{attribute 'pack_mode' := '1'} 
// ------------------------------------------------------------------------- 
//  SRCI Robot Library                                                
// ------------------------------------------------------------------------- 
//                                                                           
//  Object:      TelegramRobToPlcCyclicOptionalCartesianPosExt                                       
//  Author:      Thorsten Brach                                                
//  Date:        2024-06-01
//
//  Description:                                              
//   
//                                                                           
//  Copyright: 
//    (C) 2024 Thorsten Brach. All rights reserved                                                                         
//                                                                           
//  Disclaimer:                                                                           
//    This project is provided without any guarantee and can be used for   
//    private and commercial purposes. Any commercial use is at the user’s 
//    own risk and responsibility.
//
// -------------------------------------------------------------------------
TYPE TelegramRobToPlcCyclicOptionalCartesianPositionExt :
STRUCT
  /// Position of second external axis
  E2 : REAL;
  /// Position of third external axis
  E3 : REAL;
  /// Position of fourth external axis
  E4 : REAL;
  /// Position of fifth external axis
  E5 : REAL;
  /// Position of sixth external axis
  E6 : REAL;    
END_STRUCT
END_TYPE

{attribute 'pack_mode' := '1'} 
// ------------------------------------------------------------------------- 
//  SRCI Robot Library                                                
// ------------------------------------------------------------------------- 
//                                                                           
//  Object:      TelegramRobToPlcCyclicOptionalCurrent                                       
//  Author:      Thorsten Brach                                                
//  Date:        2024-06-01
//
//  Description:                                              
//   
//                                                                           
//  Copyright: 
//    (C) 2024 Thorsten Brach. All rights reserved                                                                         
//                                                                           
//  Disclaimer:                                                                           
//    This project is provided without any guarantee and can be used for   
//    private and commercial purposes. Any commercial use is at the user’s 
//    own risk and responsibility.
//
// -------------------------------------------------------------------------
TYPE TelegramRobToPlcCyclicOptionalCurrent :
STRUCT
  /// Current of first joint of the robot
  J1 : REAL;
  /// Current of second joint of the robot
  J2 : REAL;
  /// Current of third joint of the robot
  J3 : REAL;
  /// Current of fourth joint of the robot
  J4 : REAL;
  /// Current of fifth joint of the robot
  J5 : REAL;
  /// Current of sixth joint of the robot
  J6 : REAL;  
END_STRUCT
END_TYPE

{attribute 'pack_mode' := '1'} 
// ------------------------------------------------------------------------- 
//  SRCI Robot Library                                                
// ------------------------------------------------------------------------- 
//                                                                           
//  Object:      TelegramRobToPlcCyclicOptionalCurrentExt                                       
//  Author:      Thorsten Brach                                                
//  Date:        2024-06-01
//
//  Description:                                              
//   
//                                                                           
//  Copyright: 
//    (C) 2024 Thorsten Brach. All rights reserved                                                                         
//                                                                           
//  Disclaimer:                                                                           
//    This project is provided without any guarantee and can be used for   
//    private and commercial purposes. Any commercial use is at the user’s 
//    own risk and responsibility.
//
// -------------------------------------------------------------------------
TYPE TelegramRobToPlcCyclicOptionalCurrentExt :
STRUCT
  /// Current of first external joint of the robot
  E1 : REAL;
  /// Current of second external axis
  E2: REAL;
  /// Current of third external axis
  E3: REAL;
  /// Current of fourth external axis
  E4: REAL;
  /// Current of fifth external axis
  E5: REAL;
  /// Current of sixth external axis
  E6: REAL;  
END_STRUCT
END_TYPE

{attribute 'pack_mode' := '1'} 
// ------------------------------------------------------------------------- 
//  SRCI Robot Library                                                
// ------------------------------------------------------------------------- 
//                                                                           
//  Object:      TelegramRobToPlcCyclicOptionalForce                                       
//  Author:      Thorsten Brach                                                
//  Date:        2024-06-01
//
//  Description:                                              
//   
//                                                                           
//  Copyright: 
//    (C) 2024 Thorsten Brach. All rights reserved                                                                         
//                                                                           
//  Disclaimer:                                                                           
//    This project is provided without any guarantee and can be used for   
//    private and commercial purposes. Any commercial use is at the user’s 
//    own risk and responsibility.
//
// -------------------------------------------------------------------------
TYPE TelegramRobToPlcCyclicOptionalForce :
STRUCT
  /// Force on the X-Axis
  X : REAL;
  /// Force on the Y-Axis
  Y : REAL;
  /// Force on the Z-Axis
  Z : REAL;
  /// Force around the X-Axis (RX)
  Rx : REAL;
  /// Force around the Y-Axis (RY)
  Ry : REAL;
  /// Force around the Z-Axis (RZ)
  Rz : REAL;
END_STRUCT
END_TYPE

{attribute 'pack_mode' := '1'} 
// ------------------------------------------------------------------------- 
//  SRCI Robot Library                                                
// ------------------------------------------------------------------------- 
//                                                                           
//  Object:      TelegramRobToPlcCyclicOptionalForceExt                                       
//  Author:      Thorsten Brach                                                
//  Date:        2024-06-01
//
//  Description:                                              
//   
//                                                                           
//  Copyright: 
//    (C) 2024 Thorsten Brach. All rights reserved                                                                         
//                                                                           
//  Disclaimer:                                                                           
//    This project is provided without any guarantee and can be used for   
//    private and commercial purposes. Any commercial use is at the user’s 
//    own risk and responsibility.
//
// -------------------------------------------------------------------------
TYPE TelegramRobToPlcCyclicOptionalForceExt :
STRUCT
  /// Force on the external axis 1
  E1 : REAL;
  /// Force on the external axis 2
  E2 : REAL;
  /// Force on the external axis 3
  E3 : REAL;
  /// Force om the external axis 4
  E4 : REAL;
  /// Force on the external axis 5
  E5 : REAL;
  /// Force on the external axis 6
  E6 : REAL;
END_STRUCT
END_TYPE

{attribute 'pack_mode' := '1'} 
// ------------------------------------------------------------------------- 
//  SRCI Robot Library                                                
// ------------------------------------------------------------------------- 
//                                                                           
//  Object:      TelegramRobToPlcCyclicOptionalJointPosition                                       
//  Author:      Thorsten Brach                                                
//  Date:        2024-06-01
//
//  Description:                                              
//   
//                                                                           
//  Copyright: 
//    (C) 2024 Thorsten Brach. All rights reserved                                                                         
//                                                                           
//  Disclaimer:                                                                           
//    This project is provided without any guarantee and can be used for   
//    private and commercial purposes. Any commercial use is at the user’s 
//    own risk and responsibility.
//
// -------------------------------------------------------------------------
TYPE TelegramRobToPlcCyclicOptionalJointPosition :
STRUCT
  /// Position of first joint of the robot
  J1 : REAL;
  /// Position of second joint of the robot
  J2 : REAL;
  /// Position of third joint of the robot
  J3 : REAL;
  /// Position of fourth joint of the robot
  J4 : REAL;
  /// Position of fifth joint of the robot
  J5 : REAL;
  /// Position of sixth joint of the robot
  J6 : REAL;
  /// Position of first external axis 
  E1 : REAL;  
  /// Reserve
  E1_Reserve : WORD;
END_STRUCT
END_TYPE

{attribute 'pack_mode' := '1'} 
// ------------------------------------------------------------------------- 
//  SRCI Robot Library                                                
// ------------------------------------------------------------------------- 
//                                                                           
//  Object:      TelegramRobToPlcCyclicOptionalJointPositionExt                                       
//  Author:      Thorsten Brach                                                
//  Date:        2024-06-01
//
//  Description:                                              
//   
//                                                                           
//  Copyright: 
//    (C) 2024 Thorsten Brach. All rights reserved                                                                         
//                                                                           
//  Disclaimer:                                                                           
//    This project is provided without any guarantee and can be used for   
//    private and commercial purposes. Any commercial use is at the user’s 
//    own risk and responsibility.
//
// -------------------------------------------------------------------------
TYPE TelegramRobToPlcCyclicOptionalJointPositionExt :
STRUCT
  /// Position of second external axis
  E2: REAL;
  /// Position of third external axis
  E3: REAL;
  /// Position of fourth external axis
  E4: REAL;
  /// Position of fifth external axis
  E5: REAL;
  /// Position of sixth external axis
  E6: REAL;    
END_STRUCT
END_TYPE

{attribute 'pack_mode' := '1'} 
// ------------------------------------------------------------------------- 
//  SRCI Robot Library                                                
// ------------------------------------------------------------------------- 
//                                                                           
//  Object:      TelegramRobToPlcCyclicOptionalSubProgramData                                       
//  Author:      Thorsten Brach                                                
//  Date:        2024-06-01
//
//  Description:                                              
//   
//                                                                           
//  Copyright: 
//    (C) 2024 Thorsten Brach. All rights reserved                                                                         
//                                                                           
//  Disclaimer:                                                                           
//    This project is provided without any guarantee and can be used for   
//    private and commercial purposes. Any commercial use is at the user’s 
//    own risk and responsibility.
//
// -------------------------------------------------------------------------
TYPE TelegramRobToPlcCyclicOptionalSubProgramData :
STRUCT
  /// Sub program data
  Data : ARRAY [0..25] OF BYTE;
END_STRUCT
END_TYPE

{attribute 'pack_mode' := '1'} 
// ------------------------------------------------------------------------- 
//  SRCI Robot Library                                                
// ------------------------------------------------------------------------- 
//                                                                           
//  Object:      ActivateNextCommandOutCmd                                       
//  Author:      Thorsten Brach                                                
//  Date:        2024-06-01
//
//  Description:                                              
//   
//                                                                           
//  Copyright: 
//    (C) 2024 Thorsten Brach. All rights reserved                                                                         
//                                                                           
//  Disclaimer:                                                                           
//    This project is provided without any guarantee and can be used for   
//    private and commercial purposes. Any commercial use is at the user’s 
//    own risk and responsibility.
//
// -------------------------------------------------------------------------
TYPE ActivateNextCommandOutCmd :
STRUCT
  /// Unique system-generated ID of the "Action" when the function is triggered.
  /// • >0: The "Action" is started by the trigger function with identical FollowID.
  /// • <0: The "Action" is stopped by the trigger function with identical FollowID.
  /// For more information see chapter 5.5.12.4 EmitterID, ListenerID, FollowID and OriginID
  OriginID           : INT;
  /// Relates to ListenerID >0
  /// Number of successful trigger -based command invocations
  /// For more information refer to chapter 5.5.12.4.
  InvocationCounter  : USINT;
END_STRUCT
END_TYPE

{attribute 'pack_mode' := '1'} 
// ------------------------------------------------------------------------- 
//  SRCI Robot Library                                                
// ------------------------------------------------------------------------- 
//                                                                           
//  Object:      ActivateNextCommandParCmd                                       
//  Author:      Thorsten Brach                                                
//  Date:        2024-06-01
//
//  Description:                                              
//   
//                                                                           
//  Copyright: 
//    (C) 2024 Thorsten Brach. All rights reserved                                                                         
//                                                                           
//  Disclaimer:                                                                           
//    This project is provided without any guarantee and can be used for   
//    private and commercial purposes. Any commercial use is at the user’s 
//    own risk and responsibility.
//
// -------------------------------------------------------------------------
TYPE ActivateNextCommandParCmd :
STRUCT
  /// Processing mode
  ProcessingMode : ProcessingMode;
  /// ID of the trigger function that may be triggered:
  /// • 0: Immediately (default). - Start executing THIS function immediately.
  /// • >0: Triggero Start executing when the trigger function with the identical EmitterID is called.
  /// For more information see chapter 5.5.12.4.
  ListenerID     : SINT;
END_STRUCT
END_TYPE

{attribute 'pack_mode' := '1'} 
// ------------------------------------------------------------------------- 
//  SRCI Robot Library                                                
// ------------------------------------------------------------------------- 
//                                                                           
//  Object:      ActivateNextCommandRecvData                                       
//  Author:      Thorsten Brach                                                
//  Date:        2024-06-01
//
//  Description:                                              
//   
//                                                                           
//  Copyright: 
//    (C) 2024 Thorsten Brach. All rights reserved                                                                         
//                                                                           
//  Disclaimer:                                                                           
//    This project is provided without any guarantee and can be used for   
//    private and commercial purposes. Any commercial use is at the user’s 
//    own risk and responsibility.
//
// -------------------------------------------------------------------------
TYPE ActivateNextCommandRecvData EXTENDS RspHeader :
STRUCT
  /// Relates to ListenerID >0
  /// Number of successful trigger -based command invocations
  /// For more information refer to chapter 5.5.12.4.
  InvocationCounter  : USINT;
  /// Reserve
  Reserve            : SINT;
  /// Unique system-generated ID of the "Action" when the function is triggered.
  /// • >0: The "Action" is started by the trigger function with identical FollowID.
  /// • <0: The "Action" is stopped by the trigger function with identical FollowID.
  /// For more information see chapter 5.5.12.4 EmitterID, ListenerID, FollowID and OriginID
  OriginID           : INT;
END_STRUCT
END_TYPE

{attribute 'pack_mode' := '1'}
// ------------------------------------------------------------------------- 
//  SRCI Robot Library                                                
// ------------------------------------------------------------------------- 
//                                                                           
//  Object:      ActivateNextCommandParCmd                                       
//  Author:      Thorsten Brach                                                
//  Date:        2024-06-01
//
//  Description:                                              
//   
//                                                                           
//  Copyright: 
//    (C) 2024 Thorsten Brach. All rights reserved                                                                         
//                                                                           
//  Disclaimer:                                                                           
//    This project is provided without any guarantee and can be used for   
//    private and commercial purposes. Any commercial use is at the user’s 
//    own risk and responsibility.
//
// -------------------------------------------------------------------------
TYPE ActivateNextCommandSendData EXTENDS CmdHeader:   
STRUCT  
  /// ID of Action that will be executed when this command is active
  /// • >0: Start Action        - Start executing the Action function with the identical ListenerID.
  /// • <0: Stop Action         - Stop executing the Action function with the identical ListenerID.
  /// •  0: Undefined (default) - If no EmitterID is defined, the function returns an error message
  /// For more information see chapter 5.5.12.4
  EmitterID  : ARRAY[0..3] OF SINT;  
  /// ID of the trigger function that may be triggered:
  /// • 0: Immediately (default). - Start executing THIS function immediately.
  /// • >0: Triggero Start executing when the trigger function with the identical EmitterID is called.
  /// For more information see chapter 5.5.12.4.
  ListenerID : SINT;
  /// Reserve
  Reserve    : BYTE;
END_STRUCT
END_TYPE

{attribute 'pack_mode' := '1'} 
// ------------------------------------------------------------------------- 
//  SRCI Robot Library                                                
// ------------------------------------------------------------------------- 
//                                                                           
//  Object:      ActivateWorkAreaOutCmd                                       
//  Author:      Thorsten Brach                                                
//  Date:        2024-06-01
//
//  Description:                                              
//   
//                                                                           
//  Copyright: 
//    (C) 2024 Thorsten Brach. All rights reserved                                                                         
//                                                                           
//  Disclaimer:                                                                           
//    This project is provided without any guarantee and can be used for   
//    private and commercial purposes. Any commercial use is at the user’s 
//    own risk and responsibility.
//
// -------------------------------------------------------------------------
TYPE ActivateWorkAreaOutCmd :
STRUCT
END_STRUCT
END_TYPE

{attribute 'pack_mode' := '1'} 
// ------------------------------------------------------------------------- 
//  SRCI Robot Library                                                
// ------------------------------------------------------------------------- 
//                                                                           
//  Object:      ActivateWorkAreaParCmd                                       
//  Author:      Thorsten Brach                                                
//  Date:        2024-06-01
//
//  Description:                                              
//   
//                                                                           
//  Copyright: 
//    (C) 2024 Thorsten Brach. All rights reserved                                                                         
//                                                                           
//  Disclaimer:                                                                           
//    This project is provided without any guarantee and can be used for   
//    private and commercial purposes. Any commercial use is at the user’s 
//    own risk and responsibility.
//
// -------------------------------------------------------------------------
TYPE ActivateWorkAreaParCmd :
STRUCT
  /// Index of the robot work area to be activated
  /// • 0 (default)..254
  WorkAreaNo         : USINT;
  /// Set to activate work area defined by Index.
  /// Reset to deactivate work area defined by Index.
  ActivateArea       : BOOL;
END_STRUCT
END_TYPE

{attribute 'pack_mode' := '1'} 
// ------------------------------------------------------------------------- 
//  SRCI Robot Library                                                
// ------------------------------------------------------------------------- 
//                                                                           
//  Object:      ActivateWorkAreaRecvData                                       
//  Author:      Thorsten Brach                                                
//  Date:        2024-06-01
//
//  Description:                                              
//   
//                                                                           
//  Copyright: 
//    (C) 2024 Thorsten Brach. All rights reserved                                                                         
//                                                                           
//  Disclaimer:                                                                           
//    This project is provided without any guarantee and can be used for   
//    private and commercial purposes. Any commercial use is at the user’s 
//    own risk and responsibility.
//
// -------------------------------------------------------------------------
TYPE ActivateWorkAreaRecvData EXTENDS RspHeader :
STRUCT
END_STRUCT
END_TYPE

{attribute 'pack_mode' := '1'}
// ------------------------------------------------------------------------- 
//  SRCI Robot Library                                                
// ------------------------------------------------------------------------- 
//                                                                           
//  Object:      ActivateWorkAreaParCmd                                       
//  Author:      Thorsten Brach                                                
//  Date:        2024-06-01
//
//  Description:                                              
//   
//                                                                           
//  Copyright: 
//    (C) 2024 Thorsten Brach. All rights reserved                                                                         
//                                                                           
//  Disclaimer:                                                                           
//    This project is provided without any guarantee and can be used for   
//    private and commercial purposes. Any commercial use is at the user’s 
//    own risk and responsibility.
//
// -------------------------------------------------------------------------
TYPE ActivateWorkAreaSendData EXTENDS CmdHeader:   
STRUCT  
  /// Index of the robot work area to be activated
  /// • 0 (default)..254
  WorkAreaNo         : USINT;
  /// Set to activate work area defined by Index.
  /// Reset to deactivate work area defined by Index.
  ActivateArea       : BOOL;
END_STRUCT
END_TYPE

{attribute 'pack_mode' := '1'} 
// ------------------------------------------------------------------------- 
//  SRCI Robot Library                                                
// ------------------------------------------------------------------------- 
//                                                                           
//  Object:      BrakeTestOutCmd                                       
//  Author:      Thorsten Brach                                                
//  Date:        2024-06-01
//
//  Description:                                              
//   
//                                                                           
//  Copyright: 
//    (C) 2024 Thorsten Brach. All rights reserved                                                                         
//                                                                           
//  Disclaimer:                                                                           
//    This project is provided without any guarantee and can be used for   
//    private and commercial purposes. Any commercial use is at the user’s 
//    own risk and responsibility.
//
// -------------------------------------------------------------------------
TYPE BrakeTestOutCmd :
STRUCT
  /// Indicates the result of the brake test of the robot axes related to the brake test.
  /// • TRUE: The brake test has been realized successfully.
  /// • FALSE: The brake test failed. 
  /// See Table 6-735 for bit assignment.
  RobotAxesStatus    : RobotAxesFlags;
  /// Indicates the result of the brake test of the external robot axes related to the brake test.
  /// • TRUE: The brake test has been realized successfully.
  /// • FALSE: The brake test failed.
  /// See Table 6-735 for bit assignment.
  ExternalAxesStatus : ExternalAxesFlags;
  /// Indicates the warning messages availability related to the brake functionality of the robot axes reported by the RC.
  /// • TRUE: One or more warning messages are available.
  /// • FALSE: No warning message is available.
  /// See Table 6-735 for bit assignment.
  RobotAxesWarning   : RobotAxesFlags;
  /// Indicates the warning messages availability related to the brake functionality of the external robot axis reported by the RC.
  /// • TRUE: One or more warning messages are available.
  /// • FALSE: No warning message is available.
  /// See Table 6-735 for bit assignment.
  ExternalAxesWarning: ExternalAxesFlags;
END_STRUCT
END_TYPE

{attribute 'pack_mode' := '1'} 
// ------------------------------------------------------------------------- 
//  SRCI Robot Library                                                
// ------------------------------------------------------------------------- 
//                                                                           
//  Object:      BrakeTestParCmd                                       
//  Author:      Thorsten Brach                                                
//  Date:        2024-06-01
//
//  Description:                                              
//   
//                                                                           
//  Copyright: 
//    (C) 2024 Thorsten Brach. All rights reserved                                                                         
//                                                                           
//  Disclaimer:                                                                           
//    This project is provided without any guarantee and can be used for   
//    private and commercial purposes. Any commercial use is at the user’s 
//    own risk and responsibility.
//
// -------------------------------------------------------------------------
TYPE BrakeTestParCmd :
STRUCT
  /// Parameter which determines the behavior towards the previously sent and still active or buffered commands.
  AbortingMode       : AbortingMode;
  /// Defines which of the robot axis should be activated for the brake test.
  /// • TRUE (default): Axis activated.
  /// • FALSE: Axis deactivated.
  /// See Table 6-735 for bit assignment.
  RobotAxesActive    : RobotAxesFlags;
  /// Defines which of the external robot axis should be activated for the brake test.
  /// • TRUE: Axis activated.
  /// • FALSE (default): Axis deactivated.
  /// See Table 6-735 for bit assignment.   
  ExternalAxesActive : ExternalAxesFlags;
  /// Defines the target sequence in which the command will be executed
  SequenceFlag       : SequenceFlag;
END_STRUCT
END_TYPE

{attribute 'pack_mode' := '1'} 
// ------------------------------------------------------------------------- 
//  SRCI Robot Library                                                
// ------------------------------------------------------------------------- 
//                                                                           
//  Object:      BrakeTestRecvData                                       
//  Author:      Thorsten Brach                                                
//  Date:        2024-06-01
//
//  Description:                                              
//   
//                                                                           
//  Copyright: 
//    (C) 2024 Thorsten Brach. All rights reserved                                                                         
//                                                                           
//  Disclaimer:                                                                           
//    This project is provided without any guarantee and can be used for   
//    private and commercial purposes. Any commercial use is at the user’s 
//    own risk and responsibility.
//
// -------------------------------------------------------------------------
TYPE BrakeTestRecvData EXTENDS RspHeader :
STRUCT
  /// Indicates the result of the brake test of the robot axes related to the brake test.
  /// • TRUE: The brake test has been realized successfully.
  /// • FALSE: The brake test failed. 
  /// See Table 6-735 for bit assignment.
  RobotAxesStatus    : BYTE;
  /// Indicates the result of the brake test of the external robot axes related to the brake test.
  /// • TRUE: The brake test has been realized successfully.
  /// • FALSE: The brake test failed.
  /// See Table 6-735 for bit assignment.
  ExternalAxesStatus : BYTE;
  /// Indicates the warning messages availability related to the brake functionality of the robot axes reported by the RC.
  /// • TRUE: One or more warning messages are available.
  /// • FALSE: No warning message is available.
  /// See Table 6-735 for bit assignment.
  RobotAxesWarning   : BYTE;
  /// Indicates the warning messages availability related to the brake functionality of the external robot axis reported by the RC.
  /// • TRUE: One or more warning messages are available.
  /// • FALSE: No warning message is available.
  /// See Table 6-735 for bit assignment.
  ExternalAxesWarning: BYTE;
END_STRUCT
END_TYPE

{attribute 'pack_mode' := '1'}
// ------------------------------------------------------------------------- 
//  SRCI Robot Library                                                
// ------------------------------------------------------------------------- 
//                                                                           
//  Object:      BrakeTestSendData                                       
//  Author:      Thorsten Brach                                                
//  Date:        2024-06-01
//
//  Description:                                              
//   
//                                                                           
//  Copyright: 
//    (C) 2024 Thorsten Brach. All rights reserved                                                                         
//                                                                           
//  Disclaimer:                                                                           
//    This project is provided without any guarantee and can be used for   
//    private and commercial purposes. Any commercial use is at the user’s 
//    own risk and responsibility.
//
// -------------------------------------------------------------------------
TYPE BrakeTestSendData EXTENDS CmdHeader:   
STRUCT
  /// Defines which of the robot axis should be activated for the brake test.
  /// • TRUE (default): Axis activated.
  /// • FALSE: Axis deactivated.
  /// See Table 6-735 for bit assignment.
  RobotAxesActive    : BYTE;
  /// Defines which of the external robot axis should be activated for the brake test.
  /// • TRUE: Axis activated.
  /// • FALSE (default): Axis deactivated.
  /// See Table 6-735 for bit assignment.   
  ExternalAxesActive : BYTE; 
END_STRUCT
END_TYPE

{attribute 'pack_mode' := '1'} 
// ------------------------------------------------------------------------- 
//  SRCI Robot Library                                                
// ------------------------------------------------------------------------- 
//                                                                           
//  Object:      BrakeTestOutCmd                                       
//  Author:      Thorsten Brach                                                
//  Date:        2024-06-01
//
//  Description:                                              
//   
//                                                                           
//  Copyright: 
//    (C) 2024 Thorsten Brach. All rights reserved                                                                         
//                                                                           
//  Disclaimer:                                                                           
//    This project is provided without any guarantee and can be used for   
//    private and commercial purposes. Any commercial use is at the user’s 
//    own risk and responsibility.
//
// -------------------------------------------------------------------------
TYPE OpenBrakeOutCmd :
STRUCT
  /// TRUE when "OpenBrake" is active.
  Enabled                   : BOOL;  
  /// Indicates the brake release status of the main robot axes.
  /// • TRUE: The brake of the axis is opened.
  /// • FALSE: The brake of the axis is closed.
  /// See Table 6-735 for bit assignment
  RobotAxesBrakeReleased    : RobotAxesFlags;
  /// Indicates the brake release status of the external robot axes.
  /// • TRUE: The brake of the axis is opened.
  /// • FALSE: The brake of the axis is closed/not supported
  /// See Table 6-735 for bit assignment
  ExternalAxesBrakeReleased : ExternalAxesFlags;
END_STRUCT
END_TYPE

{attribute 'pack_mode' := '1'} 
// ------------------------------------------------------------------------- 
//  SRCI Robot Library                                                
// ------------------------------------------------------------------------- 
//                                                                           
//  Object:      OpenBrakeParCmd                                       
//  Author:      Thorsten Brach                                                
//  Date:        2024-06-01
//
//  Description:                                              
//   
//                                                                           
//  Copyright: 
//    (C) 2024 Thorsten Brach. All rights reserved                                                                         
//                                                                           
//  Disclaimer:                                                                           
//    This project is provided without any guarantee and can be used for   
//    private and commercial purposes. Any commercial use is at the user’s 
//    own risk and responsibility.
//
// -------------------------------------------------------------------------
TYPE OpenBrakeParCmd :
STRUCT
  /// Defines which brake of the robot axes must be released.
  /// • TRUE: Open the brake of the axis.
  /// • FALSE (default): Close the brake of the axis.
  RobotAxesBrakeRelease    : RobotAxesFlags;
  /// Defines which brake of the external robot axis must be released.
  /// • TRUE: Open the brake of the axis.
  /// • FALSE (default): Close the brake of the axis.
  /// See Table 6-676 for bit assignment.
  ExternalAxesBrakeRelease : ExternalAxesFlags;
END_STRUCT
END_TYPE

{attribute 'pack_mode' := '1'} 
// ------------------------------------------------------------------------- 
//  SRCI Robot Library                                                
// ------------------------------------------------------------------------- 
//                                                                           
//  Object:      BrakeTestRecvData                                       
//  Author:      Thorsten Brach                                                
//  Date:        2024-06-01
//
//  Description:                                              
//   
//                                                                           
//  Copyright: 
//    (C) 2024 Thorsten Brach. All rights reserved                                                                         
//                                                                           
//  Disclaimer:                                                                           
//    This project is provided without any guarantee and can be used for   
//    private and commercial purposes. Any commercial use is at the user’s 
//    own risk and responsibility.
//
// -------------------------------------------------------------------------
TYPE OpenBrakeRecvData EXTENDS RspHeader :
STRUCT
  /// TRUE when "OpenBrake" is active.
  Enabled                   : BYTE;  
  /// Indicates the brake release status of the main robot axes.
  /// • TRUE: The brake of the axis is opened.
  /// • FALSE: The brake of the axis is closed.
  /// See Table 6-735 for bit assignment
  RobotAxesBrakeReleased    : BYTE;
  /// Indicates the brake release status of the external robot axes.
  /// • TRUE: The brake of the axis is opened.
  /// • FALSE: The brake of the axis is closed/not supported
  /// See Table 6-735 for bit assignment
  ExternalAxesBrakeReleased : BYTE;
END_STRUCT
END_TYPE

{attribute 'pack_mode' := '1'}
// ------------------------------------------------------------------------- 
//  SRCI Robot Library                                                
// ------------------------------------------------------------------------- 
//                                                                           
//  Object:      BrakeTestSendData                                       
//  Author:      Thorsten Brach                                                
//  Date:        2024-06-01
//
//  Description:                                              
//   
//                                                                           
//  Copyright: 
//    (C) 2024 Thorsten Brach. All rights reserved                                                                         
//                                                                           
//  Disclaimer:                                                                           
//    This project is provided without any guarantee and can be used for   
//    private and commercial purposes. Any commercial use is at the user’s 
//    own risk and responsibility.
//
// -------------------------------------------------------------------------
TYPE OpenBrakeSendData EXTENDS CmdHeader:   
STRUCT
  /// Defines which brake of the robot axes must be released.
  /// • TRUE: Open the brake of the axis.
  /// • FALSE (default): Close the brake of the axis.
  RobotAxesBrakeRelease    : BYTE;
  /// Defines which brake of the external robot axis must be released.
  /// • TRUE: Open the brake of the axis.
  /// • FALSE (default): Close the brake of the axis.
  /// See Table 6-676 for bit assignment.
  ExternalAxesBrakeRelease : BYTE;
END_STRUCT
END_TYPE

{attribute 'pack_mode' := '1'} 
// ------------------------------------------------------------------------- 
//  SRCI Robot Library                                                
// ------------------------------------------------------------------------- 
//                                                                           
//  Object:      EnableRobotOutCmd                                       
//  Author:      Thorsten Brach                                                
//  Date:        2024-06-01
//
//  Description:                                              
//   
//                                                                           
//  Copyright: 
//    (C) 2024 Thorsten Brach. All rights reserved                                                                         
//                                                                           
//  Disclaimer:                                                                           
//    This project is provided without any guarantee and can be used for   
//    private and commercial purposes. Any commercial use is at the user’s 
//    own risk and responsibility.
//
// -------------------------------------------------------------------------
TYPE EnableRobotOutCmd :
STRUCT
  /// TRUE when robot is set to RA power state "Enabled"
  Enabled           : BOOL;
END_STRUCT
END_TYPE

{attribute 'pack_mode' := '1'} 
// ------------------------------------------------------------------------- 
//  SRCI Robot Library                                                
// ------------------------------------------------------------------------- 
//                                                                           
//  Object:      EnableRobotParCmd                                       
//  Author:      Thorsten Brach                                                
//  Date:        2024-06-01
//
//  Description:                                              
//   
//                                                                           
//  Copyright: 
//    (C) 2024 Thorsten Brach. All rights reserved                                                                         
//                                                                           
//  Disclaimer:                                                                           
//    This project is provided without any guarantee and can be used for   
//    private and commercial purposes. Any commercial use is at the user’s 
//    own risk and responsibility.
//
// -------------------------------------------------------------------------
TYPE EnableRobotParCmd :
STRUCT
  /// The robot will move while HoldToRun is set TRUE
  HoldToRun  : BOOL;
  /// While activated the RI state switches to interrupted when a buffered command returns Done TRUE
  /// At least one of the optional modes must be supported
  StepMode   : StepMode;
  /// Relates to StepMode 1 (Blending) and 2 (Exact stop)
  /// Start the next buffered command with the rising edge in T1 External or T2 External
  ManualStep : BOOL;  
END_STRUCT
END_TYPE

{attribute 'pack_mode' := '1'} 
// ------------------------------------------------------------------------- 
//  SRCI Robot Library                                                
// ------------------------------------------------------------------------- 
//                                                                           
//  Object:      EnableRobotRecvData                                       
//  Author:      Thorsten Brach                                                
//  Date:        2024-06-01
//
//  Description:                                              
//   
//                                                                           
//  Copyright: 
//    (C) 2024 Thorsten Brach. All rights reserved                                                                         
//                                                                           
//  Disclaimer:                                                                           
//    This project is provided without any guarantee and can be used for   
//    private and commercial purposes. Any commercial use is at the user’s 
//    own risk and responsibility.
//
// -------------------------------------------------------------------------
TYPE EnableRobotRecvData EXTENDS RspHeader :
STRUCT
  /// TRUE when robot is set to RA power state "Enabled".
  Enabled : BOOL;
END_STRUCT
END_TYPE

{attribute 'pack_mode' := '1'}
// ------------------------------------------------------------------------- 
//  SRCI Robot Library                                                
// ------------------------------------------------------------------------- 
//                                                                           
//  Object:      ActivateNextCommandParCmd                                       
//  Author:      Thorsten Brach                                                
//  Date:        2024-06-01
//
//  Description:                                              
//   
//                                                                           
//  Copyright: 
//    (C) 2024 Thorsten Brach. All rights reserved                                                                         
//                                                                           
//  Disclaimer:                                                                           
//    This project is provided without any guarantee and can be used for   
//    private and commercial purposes. Any commercial use is at the user’s 
//    own risk and responsibility.
//
// -------------------------------------------------------------------------
TYPE EnableRobotSendData EXTENDS CmdHeader: 
STRUCT
  /// Set TRUE to change RA power state to "Enabled"
 Enable          : BOOL;
 /// The robot will move while HoldToRun is set TRUE
 HoldToRun       : BOOL;
 /// While activated the RI state switches to interrupted when a buffered command returns Done TRUE
 /// At least one of the optional modes must be supported
 StepMode        : StepMode;
 /// Relates to StepMode 1 (Blending) and 2 (Exact stop)
 /// Start the next buffered command with the rising edge in T1 External or T2 External
 ManualStep      : BOOL;  
END_STRUCT
END_TYPE

{attribute 'pack_mode' := '1'} 
// ------------------------------------------------------------------------- 
//  SRCI Robot Library                                                
// ------------------------------------------------------------------------- 
//                                                                           
//  Object:      CalculateCartesianPositionOutCmd                                       
//  Author:      Thorsten Brach                                                
//  Date:        2024-06-05
//
//  Description:                                              
//   
//                                                                           
//  Copyright: 
//    (C) 2024 Thorsten Brach. All rights reserved                                                                         
//                                                                           
//  Disclaimer:                                                                           
//    This project is provided without any guarantee and can be used for   
//    private and commercial purposes. Any commercial use is at the user’s 
//    own risk and responsibility.
//
// -------------------------------------------------------------------------
TYPE CalculateCartesianPositionOutCmd :
STRUCT
  /// Index of target tool
  /// • 0: Flange (default)
  /// • 1..254: Tool frames
  TargetToolNoReturn : USINT;
  /// Index of target frame
  /// •      0: WCS
  /// • 1..254: User frames
  TargetFrameNoReturn: USINT;
  /// Calculated cartesian position
  CartesianPositionReturn  : RobotCartesianPosition;
END_STRUCT
END_TYPE

{attribute 'pack_mode' := '1'} 
// ------------------------------------------------------------------------- 
//  SRCI Robot Library                                                
// ------------------------------------------------------------------------- 
//                                                                           
//  Object:      CalculateCartesianPositionParCmd                                       
//  Author:      Thorsten Brach                                                
//  Date:        2024-06-05
//
//  Description:                                              
//   
//                                                                           
//  Copyright: 
//    (C) 2024 Thorsten Brach. All rights reserved                                                                         
//                                                                           
//  Disclaimer:                                                                           
//    This project is provided without any guarantee and can be used for   
//    private and commercial purposes. Any commercial use is at the user’s 
//    own risk and responsibility.
//
// -------------------------------------------------------------------------
TYPE CalculateCartesianPositionParCmd :
STRUCT
  /// Index of initial frame
  /// • 0: WCS (default)
  /// • 1..254: User frames
  FrameNo            : USINT;
  /// Index of target frame
  /// • 0: WCS (default)
  /// • 1..254: User frames
  TargetFrameNo          : USINT;  
  /// Robot cartesian position.
  CartesianPosition      : RobotCartesianPosition;
END_STRUCT
END_TYPE

{attribute 'pack_mode' := '1'} 
// ------------------------------------------------------------------------- 
//  SRCI Robot Library                                                
// ------------------------------------------------------------------------- 
//                                                                           
//  Object:      CalculateCartesianPositionRecvData                                       
//  Author:      Thorsten Brach                                                
//  Date:        2024-06-05
//
//  Description:                                              
//   
//                                                                           
//  Copyright: 
//    (C) 2024 Thorsten Brach. All rights reserved                                                                         
//                                                                           
//  Disclaimer:                                                                           
//    This project is provided without any guarantee and can be used for   
//    private and commercial purposes. Any commercial use is at the user’s 
//    own risk and responsibility.
//
// -------------------------------------------------------------------------
TYPE CalculateCartesianPositionRecvData EXTENDS RspHeader :
STRUCT
  /// Index of target tool
  /// • 0: Flange (default)
  /// • 1..254: Tool frames
  TargetToolNoReturn       : USINT;
  /// Index of target frame
  /// •      0: WCS
  /// • 1..254: User frames
  TargetFrameNoReturn      : USINT;
  /// Calculated cartesian position
  CartesianPositionReturn  : RobotCartesianPosition;
END_STRUCT
END_TYPE

{attribute 'pack_mode' := '1'}
// ------------------------------------------------------------------------- 
//  SRCI Robot Library                                                
// ------------------------------------------------------------------------- 
//                                                                           
//  Object:      CalculateCartesianPositionSendData                                       
//  Author:      Thorsten Brach                                                
//  Date:        2024-06-05
//
//  Description:                                              
//   
//                                                                           
//  Copyright: 
//    (C) 2024 Thorsten Brach. All rights reserved                                                                         
//                                                                           
//  Disclaimer:                                                                           
//    This project is provided without any guarantee and can be used for   
//    private and commercial purposes. Any commercial use is at the user’s 
//    own risk and responsibility.
//
// -------------------------------------------------------------------------
TYPE CalculateCartesianPositionSendData EXTENDS CmdHeader:   
STRUCT
  /// Index of source frame
  /// • 0: WCS (default)
  /// • 1..254: User frames
  FrameNo       : USINT;
  /// Index of target frame
  /// • 0: WCS (default)
  /// • 1..254: User frames
  TargetFrameNo : USINT;
  /// Robot cartesian position.
  CartesianPosition      : RobotCartesianPosition;
END_STRUCT
END_TYPE

{attribute 'pack_mode' := '1'} 
// ------------------------------------------------------------------------- 
//  SRCI Robot Library                                                
// ------------------------------------------------------------------------- 
//                                                                           
//  Object:      CalculateCartesianPositionOutCmd                                       
//  Author:      Thorsten Brach                                                
//  Date:        2024-06-05
//
//  Description:                                              
//   
//                                                                           
//  Copyright: 
//    (C) 2024 Thorsten Brach. All rights reserved                                                                         
//                                                                           
//  Disclaimer:                                                                           
//    This project is provided without any guarantee and can be used for   
//    private and commercial purposes. Any commercial use is at the user’s 
//    own risk and responsibility.
//
// -------------------------------------------------------------------------
TYPE CalculateForwardKinematicOutCmd :
STRUCT
  /// Index of target tool
  /// • 0: Flange (default)
  /// • 1..254: Tool frames
  TargetToolNoReturn : USINT;
  /// Index of target frame
  /// •      0: WCS
  /// • 1..254: User frames
  TargetFrameNoReturn: USINT;
  /// Calculated cartesian position
  CartesianPosition  : RobotCartesianPosition;
END_STRUCT
END_TYPE

{attribute 'pack_mode' := '1'} 
// ------------------------------------------------------------------------- 
//  SRCI Robot Library                                                
// ------------------------------------------------------------------------- 
//                                                                           
//  Object:      CalculateCartesianPositionParCmd                                       
//  Author:      Thorsten Brach                                                
//  Date:        2024-06-05
//
//  Description:                                              
//   
//                                                                           
//  Copyright: 
//    (C) 2024 Thorsten Brach. All rights reserved                                                                         
//                                                                           
//  Disclaimer:                                                                           
//    This project is provided without any guarantee and can be used for   
//    private and commercial purposes. Any commercial use is at the user’s 
//    own risk and responsibility.
//
// -------------------------------------------------------------------------
TYPE CalculateForwardKinematicParCmd :
STRUCT
  /// Index of target tool
  /// • 0: Flange (default)
  /// • 1..254: Tool frames
  ToolNo             : USINT;
  /// Index of target frame
  /// • 0: WCS (default)
  /// • 1..254: User frames
  FrameNo            : USINT;
  /// Calculated cartesian position
  CartesianPosition  : RobotCartesianPosition;
END_STRUCT
END_TYPE

{attribute 'pack_mode' := '1'} 
// ------------------------------------------------------------------------- 
//  SRCI Robot Library                                                
// ------------------------------------------------------------------------- 
//                                                                           
//  Object:      CalculateCartesianPositionRecvData                                       
//  Author:      Thorsten Brach                                                
//  Date:        2024-06-05
//
//  Description:                                              
//   
//                                                                           
//  Copyright: 
//    (C) 2024 Thorsten Brach. All rights reserved                                                                         
//                                                                           
//  Disclaimer:                                                                           
//    This project is provided without any guarantee and can be used for   
//    private and commercial purposes. Any commercial use is at the user’s 
//    own risk and responsibility.
//
// -------------------------------------------------------------------------
TYPE CalculateForwardKinematicRecvData EXTENDS RspHeader :
STRUCT
  /// Index of target tool
  /// • 0: Flange (default)
  /// • 1..254: Tool frames
  TargetToolNoReturn       : USINT;
  /// Index of target frame
  /// •      0: WCS
  /// • 1..254: User frames
  TargetFrameNoReturn      : USINT;
  /// Calculated cartesian position
  CartesianPosition        : RobotCartesianPosition;
END_STRUCT
END_TYPE

{attribute 'pack_mode' := '1'}
// ------------------------------------------------------------------------- 
//  SRCI Robot Library                                                
// ------------------------------------------------------------------------- 
//                                                                           
//  Object:      CalculateCartesianPositionSendData                                       
//  Author:      Thorsten Brach                                                
//  Date:        2024-06-05
//
//  Description:                                              
//   
//                                                                           
//  Copyright: 
//    (C) 2024 Thorsten Brach. All rights reserved                                                                         
//                                                                           
//  Disclaimer:                                                                           
//    This project is provided without any guarantee and can be used for   
//    private and commercial purposes. Any commercial use is at the user’s 
//    own risk and responsibility.
//
// -------------------------------------------------------------------------
TYPE CalculateForwardKinematicSendData EXTENDS CmdHeader:   
STRUCT
  /// Index of target tool
  /// • 0: Flange (default)
  /// • 1..254: Tool frames
  ToolNo             : USINT;
  /// Index of target frame
  /// • 0: WCS (default)
  /// • 1..254: User frames
  FrameNo            : USINT;
  /// Calculated cartesian position
  CartesianPosition  : RobotCartesianPosition;
END_STRUCT
END_TYPE

FUNCTION CombineHalfBytes : USINT
// ------------------------------------------------------------------------- 
//  SRCI Robot Library                                                
// ------------------------------------------------------------------------- 
//                                                                           
//  Object:      CombineHalfBytes                                       
//  Author:      Thorsten Brach                                                
//  Date:        2024-06-01
//
//  Description:                                              
//   
//                                                                           
//  Copyright: 
//    (C) 2024 Thorsten Brach. All rights reserved                                                                         
//                                                                           
//  Disclaimer:                                                                           
//    This project is provided without any guarantee and can be used for   
//    private and commercial purposes. Any commercial use is at the user’s 
//    own risk and responsibility.
//
// -------------------------------------------------------------------------
VAR_INPUT
  /// Half-Byte to add to the upper 4 Bit
  HalfByteHi : BYTE;
  /// Half-Byte to add to the lower 4 Bit
  HalfByteLo : BYTE;
END_VAR

                  // merage ParSeq and Priority to combined variable
CombineHalfBytes.0 := HalfByteLo.0;
CombineHalfBytes.1 := HalfByteLo.1;
CombineHalfBytes.2 := HalfByteLo.2;
CombineHalfBytes.3 := HalfByteLo.3;

CombineHalfBytes.4 := HalfByteHi.0;
CombineHalfBytes.5 := HalfByteHi.1;
CombineHalfBytes.6 := HalfByteHi.2;
CombineHalfBytes.7 := HalfByteHi.3;
                
END_FUNCTION

FUNCTION DATE_TO_IEC_DATE : IEC_DATE
// ------------------------------------------------------------------------- 
//  SRCI Robot Library                                                
// ------------------------------------------------------------------------- 
//                                                                           
//  Object:      DATE_TO_IEC_DATE                                       
//  Author:      Thorsten Brach                                                
//  Date:        2024-06-01
//
//  Description:                                              
//   
//                                                                           
//  Copyright: 
//    (C) 2024 Thorsten Brach. All rights reserved                                                                         
//                                                                           
//  Disclaimer:                                                                           
//    This project is provided without any guarantee and can be used for   
//    private and commercial purposes. Any commercial use is at the user’s 
//    own risk and responsibility.
//
// -------------------------------------------------------------------------
VAR_INPUT
  Value    : DATE;
END_VAR

VAR
 _tmpDate1 : DWORD;
 _tmpDate2 : DWORD;
 _initDate : DATE := DATE#1990-01-01;
END_VAR

                  /// copy date to dword
MemCpy( ADR(_tmpDate1), ADR( Value   ), SIZEOF( Value   ));
/// copy date to dword
MemCpy( ADR(_tmpDate2), ADR(_initDate), SIZEOF(_initDate));
/// calculate IEC Date
DATE_TO_IEC_DATE := DWORD_TO_USINT(_tmpDate1 - _tmpDate2); {warning 'ToDo: Check if the result is Siemens IEC Date'}
                
END_FUNCTION

FUNCTION DwordToRaStatusWord : RaStatusWord
VAR_INPUT
  /// Value
  Value : DWORD;
END_VAR

                  DwordToRaStatusWord.IsMoving                 := Value.00;
DwordToRaStatusWord.PrimarySequencePaused    := Value.01;
DwordToRaStatusWord.InPrimaryPos             := Value.02;
DwordToRaStatusWord.SecondarySequenceActive  := Value.03;
DwordToRaStatusWord.IsBlending               := Value.04;
DwordToRaStatusWord.ErrorPending             := Value.05;
DwordToRaStatusWord.RestartInProgress        := Value.06;
DwordToRaStatusWord.Enabled                  := Value.07;
DwordToRaStatusWord.Executing                := Value.08;
DwordToRaStatusWord.Interrupted              := Value.09;
DwordToRaStatusWord.OperationMode.0          := Value.10;
DwordToRaStatusWord.OperationMode.1          := Value.11;
DwordToRaStatusWord.OperationMode.2          := Value.12;
DwordToRaStatusWord.CollisionDetectedEnabled := Value.13;
DwordToRaStatusWord.CollisionDetected        := Value.14;
DwordToRaStatusWord.RestartRequested         := Value.15;
DwordToRaStatusWord.Accelerating             := Value.16;
DwordToRaStatusWord.Decelerating             := Value.17;
DwordToRaStatusWord.ConstantVelocity         := Value.18;
DwordToRaStatusWord.Bit19                    := Value.19;
DwordToRaStatusWord.Bit20                    := Value.20;
DwordToRaStatusWord.Bit21                    := Value.21;
DwordToRaStatusWord.Bit22                    := Value.22;
DwordToRaStatusWord.Bit23                    := Value.23;
DwordToRaStatusWord.Bit24                    := Value.24;
DwordToRaStatusWord.Bit25                    := Value.25;
DwordToRaStatusWord.Bit26                    := Value.26;
DwordToRaStatusWord.Bit27                    := Value.27;
DwordToRaStatusWord.Bit28                    := Value.28;
DwordToRaStatusWord.Bit29                    := Value.29;
DwordToRaStatusWord.Bit30                    := Value.30;
DwordToRaStatusWord.Bit31                    := Value.31;
                
END_FUNCTION

FUNCTION FragmentActionToByte : BYTE
// ------------------------------------------------------------------------- 
//  SRCI Robot Library                                                
// ------------------------------------------------------------------------- 
//                                                                           
//  Object:      FragmentActionToByte                                       
//  Author:      Thorsten Brach                                                
//  Date:        2024-06-01
//
//  Description:                                              
//   
//                                                                           
//  Copyright: 
//    (C) 2024 Thorsten Brach. All rights reserved                                                                         
//                                                                           
//  Disclaimer:                                                                           
//    This project is provided without any guarantee and can be used for   
//    private and commercial purposes. Any commercial use is at the user’s 
//    own risk and responsibility.
//
// -------------------------------------------------------------------------
VAR_INPUT
  FragmentAction : FragmentAction;
END_VAR

                  FragmentActionToByte.0 := FragmentAction.Complete;
FragmentActionToByte.1 := FragmentAction.Reset;
FragmentActionToByte.2 := FragmentAction.Complete;
FragmentActionToByte.3 := FragmentAction.BIT03;
FragmentActionToByte.4 := FragmentAction.BIT04;
FragmentActionToByte.5 := FragmentAction.BIT05;
FragmentActionToByte.6 := FragmentAction.BIT06;
FragmentActionToByte.7 := FragmentAction.BIT07;
                
END_FUNCTION

FUNCTION SwapBytes 
// ------------------------------------------------------------------------- 
//  SRCI Robot Library                                                
// ------------------------------------------------------------------------- 
//                                                                           
//  Object:      SwapBytes                                       
//  Author:      Thorsten Brach                                                
//  Date:        2024-06-01
//
//  Description:                                              
//   
//                                                                           
//  Copyright: 
//    (C) 2024 Thorsten Brach. All rights reserved                                                                         
//                                                                           
//  Disclaimer:                                                                           
//    This project is provided without any guarantee and can be used for   
//    private and commercial purposes. Any commercial use is at the user’s 
//    own risk and responsibility.
//
// -------------------------------------------------------------------------
VAR_INPUT
  /// pointer to data type
  pValue : POINTER TO BYTE;
  /// size of data type
  Size  : UDINT;
END_VAR

VAR
  /// Pointer to low word low byte
  _pLwLb    : POINTER TO BYTE;
  /// Pointer to low word high byte
  _pLwHb    : POINTER TO BYTE;
  /// Pointer to high word low byte
  _pHwLb    : POINTER TO BYTE;
  /// Pointer to high word high byte
  _pHwHb    : POINTER TO BYTE;  
   /// temporary bytes
  _tmpBytes : ARRAY[1..4] OF BYTE;  
END_VAR

                  IF ( RobotLibraryParameter.SWAP_BYTE_ORDER AND Size = 2)
THEN
 _pLwLb := pValue + 0;
 _pLwHb := pValue + 1;
  
  // swap bytes
 _tmpBytes[1] := _pLwHb^;
 _tmpBytes[2] := _pLwLb^;
  
  // copy bytes to data type
  MemCpy(pValue, ADR(_tmpBytes), Size);
END_IF


IF ( RobotLibraryParameter.SWAP_BYTE_ORDER AND Size = 4)
THEN
 _pLwLb := pValue + 0;
 _pLwHb := pValue + 1;
 _pHwLb := pValue + 2;
 _pHwHb := pValue + 3;
  
  // swap bytes
 _tmpBytes[1] := _pHwHb^;
 _tmpBytes[2] := _pHwLb^;
 _tmpBytes[3] := _pLwHb^;
 _tmpBytes[4] := _pLwLb^;
  
  // copy bytes to data type
  MemCpy(pValue, ADR(_tmpBytes),Size);  
END_IF
                
END_FUNCTION

FUNCTION SwapDword : DWORD
// ------------------------------------------------------------------------- 
//  SRCI Robot Library                                                
// ------------------------------------------------------------------------- 
//                                                                           
//  Object:      SwapDword                                       
//  Author:      Thorsten Brach                                                
//  Date:        2024-06-01
//
//  Description:                                              
//   
//                                                                           
//  Copyright: 
//    (C) 2024 Thorsten Brach. All rights reserved                                                                         
//                                                                           
//  Disclaimer:                                                                           
//    This project is provided without any guarantee and can be used for   
//    private and commercial purposes. Any commercial use is at the user’s 
//    own risk and responsibility.
//
// -------------------------------------------------------------------------
VAR_INPUT
  /// Value
  Value : DWORD;
END_VAR

                  SwapBytes(ADR(Value),SIZEOF(Value));

SwapDword := Value;
                
END_FUNCTION

FUNCTION SwapInt : INT
// ------------------------------------------------------------------------- 
//  SRCI Robot Library                                                
// ------------------------------------------------------------------------- 
//                                                                           
//  Object:      SwapInt                                       
//  Author:      Thorsten Brach                                                
//  Date:        2024-06-01
//
//  Description:                                              
//   
//                                                                           
//  Copyright: 
//    (C) 2024 Thorsten Brach. All rights reserved                                                                         
//                                                                           
//  Disclaimer:                                                                           
//    This project is provided without any guarantee and can be used for   
//    private and commercial purposes. Any commercial use is at the user’s 
//    own risk and responsibility.
//
// -------------------------------------------------------------------------
VAR_INPUT
  /// Value to swap
  Value : INT;
END_VAR

                  SwapBytes(ADR(Value),SIZEOF(Value));

SwapInt := Value;
                
END_FUNCTION

FUNCTION SwapReal : REAL
// ------------------------------------------------------------------------- 
//  SRCI Robot Library                                                
// ------------------------------------------------------------------------- 
//                                                                           
//  Object:      SwapReal                                       
//  Author:      Thorsten Brach                                                
//  Date:        2024-06-01
//
//  Description:                                              
//   
//                                                                           
//  Copyright: 
//    (C) 2024 Thorsten Brach. All rights reserved                                                                         
//                                                                           
//  Disclaimer:                                                                           
//    This project is provided without any guarantee and can be used for   
//    private and commercial purposes. Any commercial use is at the user’s 
//    own risk and responsibility.
//
// -------------------------------------------------------------------------
VAR_INPUT
  /// Value
  Value : REAL;
END_VAR

                  SwapBytes(ADR(Value),SIZEOF(Value));

SwapReal := Value;
                
END_FUNCTION

FUNCTION SwapTime : TOD
// ------------------------------------------------------------------------- 
//  SRCI Robot Library                                                
// ------------------------------------------------------------------------- 
//                                                                           
//  Object:      SwapTime                                       
//  Author:      Thorsten Brach                                                
//  Date:        2024-06-01
//
//  Description:                                              
//   
//                                                                           
//  Copyright: 
//    (C) 2024 Thorsten Brach. All rights reserved                                                                         
//                                                                           
//  Disclaimer:                                                                           
//    This project is provided without any guarantee and can be used for   
//    private and commercial purposes. Any commercial use is at the user’s 
//    own risk and responsibility.
//
// -------------------------------------------------------------------------
VAR_INPUT
  /// Value
  Value : TOD;
END_VAR

                  SwapBytes(ADR(Value),SIZEOF(Value));

SwapTime := Value;
                
END_FUNCTION

FUNCTION SwapUdint : UDINT
// ------------------------------------------------------------------------- 
//  SRCI Robot Library                                                
// ------------------------------------------------------------------------- 
//                                                                           
//  Object:      SwapUdint                                       
//  Author:      Thorsten Brach                                                
//  Date:        2024-06-01
//
//  Description:                                              
//   
//                                                                           
//  Copyright: 
//    (C) 2024 Thorsten Brach. All rights reserved                                                                         
//                                                                           
//  Disclaimer:                                                                           
//    This project is provided without any guarantee and can be used for   
//    private and commercial purposes. Any commercial use is at the user’s 
//    own risk and responsibility.
//
// -------------------------------------------------------------------------
VAR_INPUT
  /// Value
  Value : UDINT;
END_VAR

                  SwapBytes(ADR(Value),SIZEOF(Value));

SwapUdint := Value;
                
END_FUNCTION

FUNCTION SwapUint : UINT
// ------------------------------------------------------------------------- 
//  SRCI Robot Library                                                
// ------------------------------------------------------------------------- 
//                                                                           
//  Object:      SwapUint                                       
//  Author:      Thorsten Brach                                                
//  Date:        2024-06-01
//
//  Description:                                              
//   
//                                                                           
//  Copyright: 
//    (C) 2024 Thorsten Brach. All rights reserved                                                                         
//                                                                           
//  Disclaimer:                                                                           
//    This project is provided without any guarantee and can be used for   
//    private and commercial purposes. Any commercial use is at the user’s 
//    own risk and responsibility.
//
// -------------------------------------------------------------------------
VAR_INPUT
  /// Value to swap
  Value : UINT;
END_VAR

                  SwapBytes(ADR(Value),SIZEOF(Value));

SwapUint := Value;
                
END_FUNCTION

FUNCTION SwapWord : WORD
// ------------------------------------------------------------------------- 
//  SRCI Robot Library                                                
// ------------------------------------------------------------------------- 
//                                                                           
//  Object:      SwapWord                                       
//  Author:      Thorsten Brach                                                
//  Date:        2024-06-01
//
//  Description:                                              
//   
//                                                                           
//  Copyright: 
//    (C) 2024 Thorsten Brach. All rights reserved                                                                         
//                                                                           
//  Disclaimer:                                                                           
//    This project is provided without any guarantee and can be used for   
//    private and commercial purposes. Any commercial use is at the user’s 
//    own risk and responsibility.
//
// -------------------------------------------------------------------------
VAR_INPUT
  /// Value to swap
  Value : UINT;
END_VAR

                  SwapBytes(ADR(Value),SIZEOF(Value));

SwapWord := Value;
                
END_FUNCTION

FUNCTION TIME_TO_IEC_TIME : IEC_TIME
// ------------------------------------------------------------------------- 
//  SRCI Robot Library                                                
// ------------------------------------------------------------------------- 
//                                                                           
//  Object:      TIME_TO_IEC_TIME                                       
//  Author:      Thorsten Brach                                                
//  Date:        2024-06-01
//
//  Description:                                              
//   
//                                                                           
//  Copyright: 
//    (C) 2024 Thorsten Brach. All rights reserved                                                                         
//                                                                           
//  Disclaimer:                                                                           
//    This project is provided without any guarantee and can be used for   
//    private and commercial purposes. Any commercial use is at the user’s 
//    own risk and responsibility.
//
// -------------------------------------------------------------------------
VAR_INPUT
  Value : TOD;
END_VAR

VAR
  test : DT;
END_VAR

                  TIME_TO_IEC_TIME := Value; {warning 'ToDo: Check if the result is Siemens IEC Time'}
                
END_FUNCTION

FUNCTION VersionToByte : BYTE
// ------------------------------------------------------------------------- 
//  SRCI Robot Library                                                
// ------------------------------------------------------------------------- 
//                                                                           
//  Object:      VersionToByte                                       
//  Author:      Thorsten Brach                                                
//  Date:        2024-06-01
//
//  Description:                                              
//   
//                                                                           
//  Copyright: 
//    (C) 2024 Thorsten Brach. All rights reserved                                                                         
//                                                                           
//  Disclaimer:                                                                           
//    This project is provided without any guarantee and can be used for   
//    private and commercial purposes. Any commercial use is at the user’s 
//    own risk and responsibility.
//
// -------------------------------------------------------------------------
VAR_INPUT
  /// Version
  Value : VersionStruct;
END_VAR

VAR
  _tmpByte : BYTE;
END_VAR

                  // Minor version  • Features
//                • 0..31 minor versions
VersionToByte.0 := Value.MinorVersion.0;
VersionToByte.1 := Value.MinorVersion.1;
VersionToByte.2 := Value.MinorVersion.2;
VersionToByte.3 := Value.MinorVersion.3;
VersionToByte.4 := Value.MinorVersion.4;

// Major version  • Breaking change
//                • 0..7 major versions
VersionToByte.5 := Value.MajorVersion.0;
VersionToByte.6 := Value.MajorVersion.1;
VersionToByte.7 := Value.MajorVersion.2;
                
END_FUNCTION

FUNCTION_BLOCK RobotLibraryBaseFB
// ------------------------------------------------------------------------- 
//  SRCI Robot Library                                                
// ------------------------------------------------------------------------- 
//                                                                           
//  Object:      RobotLibraryBaseFB                                       
//  Author:      Thorsten Brach                                                
//  Date:        2024-06-01
//
//  Description:                                              
//   
//                                                                           
//  Copyright: 
//    (C) 2024 Thorsten Brach. All rights reserved                                                                         
//                                                                           
//  Disclaimer:                                                                           
//    This project is provided without any guarantee and can be used for   
//    private and commercial purposes. Any commercial use is at the user’s 
//    own risk and responsibility.
//
// -------------------------------------------------------------------------
VAR_INPUT
  /// User defined command name
  Name         : STRING(20);
END_VAR
VAR_OUTPUT
  /// Command data
  CommandData  : SendData;
  /// response data
  ResponseData : RecvData;
  /// An error occurred during the execution of the command
  Error        : BOOL;
  /// ErrorID reported by RC for error identification according to Table 7-1
  ErrorID      : WORD;
  /// WarningID for warning identification reported during execution of command according to Table 7-3
  WarningID    : WORD;
  /// InfoID for info identification reported during execution of command according to Table 7-5
  InfoID       : WORD;    
END_VAR
VAR_IN_OUT
  /// Robot assignment of function
  AxesGroup    : AxesGroup; 
END_VAR

VAR
  /// unique ID
 _uniqueID         : UDINT;  
  /// flag for response received
 _responseReceived : BOOL;
  /// internal step counter
 _stepCmd          : DINT;
  /// internal timer 
 _timerCmd         : TON;
  /// internal timeout 
 _timeoutCmd       : TIME := T#5S;


  /// internal command header
 _cmdHeader        : CmdHeader;  
  /// internal response header
 _rspHeader        : RspHeader;

END_VAR

                  OnCall      (AxesGroup := AxesGroup);
OnlineChange(AxesGroup := AxesGroup);
                

METHOD PUBLIC CallBack : DINT
VAR_INPUT
  /// Response data
  RspData : AxesGroupAcyclicAcrEntryRspBuffer;  
END_VAR
                        ResponseData.Payload    := RspData.Payload; 
ResponseData.PayloadLen := RspData.PayloadLen;
ParseResponseData(ResponseData);

// set flag for response received
_responseReceived := TRUE;
                      
END_METHOD

METHOD CheckParameterChanged : BOOL
VAR_INPUT
END_VAR
                        
                      
END_METHOD

METHOD CheckTimeout : DINT
VAR_INPUT
  /// Reference to TON instance
  rTimer : REFERENCE TO TON;
END_VAR
                        // Call timer 
rTimer();

// check if timer elapsed
IF (rTimer.Q = TRUE)
THEN
  // assign return value
  CheckTimeout := RobotLibraryConstants.OK;
ELSE
  // assign return value
  CheckTimeout := RobotLibraryConstants.RUNNING;
END_IF
                      
END_METHOD

METHOD CreateCommandData : SendData
                        // Reset all variables
CreateCommandData.Reset();
// Add CmdType
CreateCommandData.AddUint(_cmdHeader.CmdTyp);
// Add Reserve_ExecMode
CreateCommandData.AddHalfBytes(  0               , _cmdHeader.ExecMode);
// Add ParSeq_Priority
CreateCommandData.AddHalfBytes( _cmdHeader.ParSeq, _cmdHeader.Priority);
                      
END_METHOD

METHOD PROTECTED OnCall
VAR_IN_OUT
  /// Robot assignment of function
  AxesGroup         : AxesGroup; 
END_VAR
                        
                      
END_METHOD

METHOD OnlineChange : DINT
VAR
  /// Online change detected 
  OnlineChangeDetected : BOOL; {warning 'ToDo : Detect online change' }
END_VAR

VAR_IN_OUT
  /// Robot assignment of function
  AxesGroup            : AxesGroup; 
END_VAR
                        IF ( OnlineChangeDetected )
THEN
  // update reference to command FB
  AxesGroup.Acyclic.ActiveCommandRegister.OnlineChange( UniqueID := _uniqueID, rCommandFB := THIS^);
  // reset Bit for online change detected
  OnlineChangeDetected := FALSE;
END_IF
                      
END_METHOD

METHOD ParseResponseData : DINT
VAR_INPUT
  /// Response data
  ResponseData : RecvData;
END_VAR
                        // reset message IDs 
InfoID    := 0;
WarningID := 0;
ErrorID   := 0;
// reset payload pointer 
ResponseData.ResetPointer();
// get State
_rspHeader.State                := ResponseData.GetHalfeByte1(IncPayloadPtr := FALSE);
// get ParSeq
_rspHeader.ParSeq               := ResponseData.GetHalfeByte2(IncPayloadPtr := TRUE);
// get AlarmMessageSeverity
_rspHeader.AlarmMessageSeverity := ResponseData.GetByte();
// get AlarmMessageCode
_rspHeader.AlarmMessageCode     := ResponseData.GetUint();


// Update InfoID / WarningID / ErrorID
CASE _rspHeader.AlarmMessageSeverity OF

  // Informative message
  Severity.INFO        : InfoID    := _rspHeader.AlarmMessageCode;
  // Warning message
  Severity.WARNING     : WarningID := _rspHeader.AlarmMessageCode;
  // Error message
  Severity.ERROR       : ErrorID   := _rspHeader.AlarmMessageCode; 
  // Fataö error message
  Severity.FATAL_ERROR : ErrorID   := _rspHeader.AlarmMessageCode;

END_CASE
                      
END_METHOD

METHOD SetTimeout : DINT
VAR_INPUT
  /// Timeout to be set
  PT     : TIME;
  /// Reference to TON instance
  rTimer : REFERENCE TO TON;
END_VAR
                        rTimer(IN := FALSE);          // Reset timer
rTimer(PT := PT, IN := TRUE); // Start timer

// assign return value
SetTimeout := RobotLibraryConstants.OK;
                      
END_METHOD

PROPERTY NotifyParameterChanged : BOOL
GET
VAR
END_VAR
                          NotifyParameterChanged := CheckParameterChanged();
                        
END_GET
END_PROPERTY
END_FUNCTION_BLOCK

/// Handles multiple mechanisms required for operation of the interface.
FUNCTION_BLOCK RobotTaskFB
// ------------------------------------------------------------------------- 
//  SRCI Robot Library                                                
// ------------------------------------------------------------------------- 
//                                                                           
//  Object:      RobotTaskFB                                       
//  Author:      Thorsten Brach                                                
//  Date:        2024-06-01
//
//  Description:                                              
//   
//                                                                           
//  Copyright: 
//    (C) 2024 Thorsten Brach. All rights reserved                                                                         
//                                                                           
//  Disclaimer:                                                                           
//    This project is provided without any guarantee and can be used for   
//    private and commercial purposes. Any commercial use is at the user’s 
//    own risk and responsibility.
//
// -------------------------------------------------------------------------
VAR_INPUT
  /// Set TRUE (default) to initialize the interface
  Enable            : BOOL;
  /// User defined robot name
  RobotName         : STRING(20);
END_VAR

VAR_IN_OUT
  /// Inputs of PLC for communication from RC
  RobotInData       : ARRAY[1..RobotLibraryParameter.ROBOT_IN_DATA_MAX ] OF BYTE;
  /// Outputs of PLC for communication to RC
  RobotOutData      : ARRAY[1..RobotLibraryParameter.ROBOT_OUT_DATA_MAX] OF BYTE;
  ///  User data stored on the PLC according to Table 6-10
  UserData          : UserData;
  /// ToolData stored on PLC. For more information refer to 5.5.6.3
  ToolData          : ARRAY[1..RobotLibraryParameter.TOOL_MAX      ] OF ToolData;
  /// LoadData stored on PLC.For more information refer to 5.5.6.4
  FrameData         : ARRAY[1..RobotLibraryParameter.FRAME_MAX     ] OF FrameData;
  /// LoadData stored on PLC.For more information refer to 5.5.6.4
  LoadData          : ARRAY[1..RobotLibraryParameter.LOAD_MAX      ] OF LoadData;
  /// Work areas stored on PLC. For more information refer to 5.5.8
  WorkAreas         : ARRAY[1..RobotLibraryParameter.WORK_AREAS_MAX] OF RobotWorkArea;
  /// Software limits stored on PLC
  SoftwareLimits    : SWLimits;
  /// Default dynamics stored on PLC. For more information refer to 5.5.7
  DefaultDynamics   : DefaultDynamics;
  /// Reference dynamics stored on PLC. For more information refer to 5.5.7
  ReferenceDynamics : ReferenceDynamics;
  /// System log on PLC
  SystemLog         : ARRAY[1..RobotLibraryParameter.SYSTEM_LOG_MAX ] OF STRING;
  ///Message buffer on the PLC - For more information refer to 5.5.11
  MessageLog        : ARRAY[1..RobotLibraryParameter.MESSAGE_LOG_MAX] OF AlarmMessage;
  /// Robot assignment of function
  AxesGroup         : AxesGroup;
END_VAR

VAR_OUTPUT
  /// FB is being processed
  Busy              : BOOL;
  /// Interface is initialized (RI state: "Initialized").
  /// For more information on RI states refer to chapter 5.5.3.1.
  Initialized       : BOOL;
  /// Server and client were successfully synchronized (RI state: "Synchronized).
  /// For more information on the synchronization mechanism refer to chapter 5.6.7.
  Synchronized      : BOOL;
  /// An error occurred
  Error             : BOOL;
  /// ErrorID reported by RC for error identification according to Table 7-1.
  ErrorID           : WORD;
  /// WarningID for warning identification reported during execution of command according to Table 7-3.
  WarningID         : WORD;
  /// InfoID for info identification reported during execution of command according to Table 7-5.
  InfoID            : WORD;
END_VAR

VAR
  /// Execution order lost
  ExecutionOrderList : ARRAY [1..RobotLibraryParameter.ACTIVE_CMD_REGISTER_ENTRIES_MAX] OF DINT;  
  /// Send Buffer
  SendData           : SendData;
  /// Recv Buffer
  RecvData           : RecvData;
  /// Telegram 
  Telegram           : Telegram;
END_VAR

                  OnCall            (AxesGroup    := AxesGroup);

CmdManagementLayer(AxesGroup    := AxesGroup);

NetworkLayer     ( AxesGroup    := AxesGroup,
                   RobotInData  := RobotInData,
                   RobotOutData := RobotOutData);
                   
TransportLayer   ( AxesGroup    := AxesGroup);
                   
                

METHOD CmdManagementLayer : BOOL
VAR_IN_OUT
  /// Robot assignment of function
  AxesGroup : AxesGroup;
END_VAR

VAR
  /// internal index
 _idx     : DINT;  
END_VAR
                        FOR _idx := 1 TO RobotLibraryParameter.ACTIVE_CMD_REGISTER_ENTRIES_MAX
DO
  // Check reference to command FB is valid ? 
  IF ( NOT __ISVALIDREF(AxesGroup.Acyclic.ActiveCommandRegister.Register[_idx].rCommandFB))
  THEN
    RETURN;
	END_IF

  // Check Cmd Parameter changed ? 
  IF ( AxesGroup.Acyclic.ActiveCommandRegister.Register[_idx].rCommandFB.NotifyParameterChanged )
  THEN
    IF (( AxesGroup.Acyclic.ActiveCommandRegister.Register[_idx].Command[1].State <> BufferStateCmd.SENDING   ) AND
        ( AxesGroup.Acyclic.ActiveCommandRegister.Register[_idx].Command[1].State <> BufferStateCmd.PROCESSED ))
    THEN
      // add to send register
      AxesGroup.Acyclic.ActiveCommandRegister.Register[_idx].Command[1].State      := BufferStateCmd.UPDATE_AVAILABLE;
      AxesGroup.Acyclic.ActiveCommandRegister.Register[_idx].Command[1].Payload    := AxesGroup.Acyclic.ActiveCommandRegister.Register[_idx].rCommandFB.CommandData.Payload;
      AxesGroup.Acyclic.ActiveCommandRegister.Register[_idx].Command[1].PayloadLen := AxesGroup.Acyclic.ActiveCommandRegister.Register[_idx].rCommandFB.CommandData.PayloadLen;
    ELSE
      // add to buffer register
      AxesGroup.Acyclic.ActiveCommandRegister.Register[_idx].Command[2].State      := BufferStateCmd.UPDATE_AVAILABLE;
      AxesGroup.Acyclic.ActiveCommandRegister.Register[_idx].Command[2].Payload    := AxesGroup.Acyclic.ActiveCommandRegister.Register[_idx].rCommandFB.CommandData.Payload;
      AxesGroup.Acyclic.ActiveCommandRegister.Register[_idx].Command[2].PayloadLen := AxesGroup.Acyclic.ActiveCommandRegister.Register[_idx].rCommandFB.CommandData.PayloadLen;
		END_IF
  END_IF
  
  // Check Response received ? 
  IF ( AxesGroup.Acyclic.ActiveCommandRegister.Register[_idx].Response[1].State = BufferStateRsp.RECEIVED)
  THEN
    // update state
    AxesGroup.Acyclic.ActiveCommandRegister.Register[_idx].Response[1].State := BufferStateRsp.PROCESSED;
    // callback CommandFB    
    AxesGroup.Acyclic.ActiveCommandRegister.Register[_idx].rCommandFB.CallBack(AxesGroup.Acyclic.ActiveCommandRegister.Register[_idx].Response[1]);    
	END_IF

  // delete entries with State.IS_Final 
  IF ( AxesGroup.Acyclic.ActiveCommandRegister.Register[_idx].State  = ActiveCommandRegisterState.IS_FINAL )
  THEN
    MemSet(ADR(AxesGroup.Acyclic.ActiveCommandRegister.Register[_idx]), 0, SIZEOF(AxesGroup.Acyclic.ActiveCommandRegister.Register[_idx]));
	END_IF
 
END_FOR
                      
END_METHOD

METHOD CreateSendData : DINT
VAR_IN_OUT
  /// Robot assignment of function
  AxesGroup         : AxesGroup;
    /// Inputs of PLC for communication from RC
  RobotInData       : ARRAY[1..RobotLibraryParameter.ROBOT_IN_DATA_MAX ] OF BYTE;
  /// Outputs of PLC for communication to RC
  RobotOutData      : ARRAY[1..RobotLibraryParameter.ROBOT_OUT_DATA_MAX] OF BYTE;
END_VAR

VAR 
  /// internal index
 _idx        : DINT;
  /// temporary byte
 _tmpByte    : BYTE;
  /// internal register indec
 _regIdx     : DINT;
  /// internal payload pointer
 _payLoadPtr : DWORD;  
END_VAR
                        AxesGroup.Config.PlcToRob.Header.SRCIVersion               := RobotLibraryConstants.SRCIVersion;
AxesGroup.Config.PlcToRob.Header.FastStop                  := AxesGroup.Config.PlcToRob.Header.FastStop; 
AxesGroup.Config.PlcToRob.Header.LifeSign                  := AxesGroup.Config.RobToPlc.Header.LifeSign;
AxesGroup.Config.PlcToRob.Header.TelegramLengthPlcToRob    := RobotLibraryParameter.ROBOT_OUT_DATA_MAX;
AxesGroup.Config.PlcToRob.Header.TelegramLengthRobToPlc    := RobotLibraryParameter.ROBOT_IN_DATA_MAX;
AxesGroup.Config.PlcToRob.Header.AxesGroupID               := AxesGroup.Config.PlcToRob.Header.AxesGroupID;
AxesGroup.Config.PlcToRob.Header.Control                   := AxesGroup.Config.PlcToRob.Header.Control;
AxesGroup.Config.PlcToRob.Header.Reserved                  := 0;

